Staubli VAL3: onEditItem.pgx

public program onEditItem(string& x_sEvent[], num x_nIndex, num x_nIndexItem)
begin
  // edit the custom element that was add in the list
end
